Fanuc KAREL source: kc00020.KL

-- PROVISIONAL review KL for V1013-1; original PC SHA256 81c1f44810c7d5092cd4427dcdb7493e63aff143960533d6df9200a2dbe3f32e
-- Incomplete behavior may be omitted. Consult companion uncertainty JSON. Do not deploy.
PROGRAM KC00020
%NOLOCKGROUP
BEGIN
  -- UNRESOLVED_PC offsets 5-12; opcodes 27,27,27,9C,31
  -- UNRESOLVED_PC offsets 17-21; opcodes 7F
END KC00020
